PROGRAM MAIN
VAR
bEnable: BOOL
bStart: BOOL 
END_VAR

bEnable:=bStart

END_PROGRAM

(* stored: Version 1.1.0.1, ProductVersion 3.1.4024.12
   POU MAIN: Id {a15ca992-4d0c-4d04-b312-e218ff3c5355}, SpecialFunc None *)
